// TIA Portal V17 export
// export: Created 2025-03-07T09:16:44.2659713Z, ExportSetting WithDefaults, DisplayName Totally Integrated Automation Portal, DisplayVersion V17 Update 8, DisplayName TIA Portal Openness, DisplayVersion V17 Update 8, DisplayName TIA Portal Version Control Interface, DisplayVersion V17, DisplayName SINAMICS Startdrive Advanced, DisplayVersion V17 SP2, DisplayName SINAMICS Startdrive G110M, G120, G120C, G120D, G120P, G115D, DisplayVersion V17 SP2, DisplayName SINAMICS Startdrive G130, G150, S120, S150, SINAMICS MV, S210, DisplayVersion V17 SP2, DisplayName STEP 7 Professional, DisplayVersion V17 Update 8, DisplayName SINUMERIK ONE STEP 7 Toolbox, DisplayVersion V17 Update 12, DisplayName SINUMERIK 840D sl STEP 7 Toolbox, DisplayVersion V17 Update 12, DisplayName STEP 7 Safety, DisplayVersion V17 Update 6, DisplayName WinCC Advanced, DisplayVersion V17 Update 8
FUNCTION "FC3001_JAW_CHUCK_CONTROL_U01_STA_1" : Void   // FC3001, LAD
{ S7_Optimized_Access := 'TRUE' }
VERSION : 0.1
// stored: AutoNumber false, IsIECCheckEnabled false, SetENOAutomatically false, UDAEnableTagReadback false
   VAR_TEMP
      TEMP_SENSOR_VALUE_1 : UInt;
      TEMP_SENSOR_VALUE : UInt;
   END_VAR
BEGIN

REGION Network 1: INPUTS
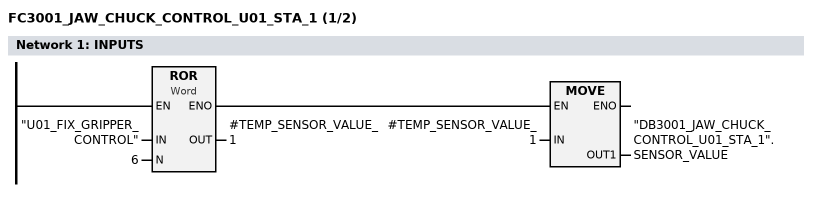
   #TEMP_SENSOR_VALUE_1 := ROR(IN := "U01_FIX_GRIPPER_CONTROL", N := 6);
   "DB3001_JAW_CHUCK_CONTROL_U01_STA_1".SENSOR_VALUE := #TEMP_SENSOR_VALUE_1;
END_REGION

REGION Network 2: UNIT 01 STATION 1 FIXTURE CLAMPED
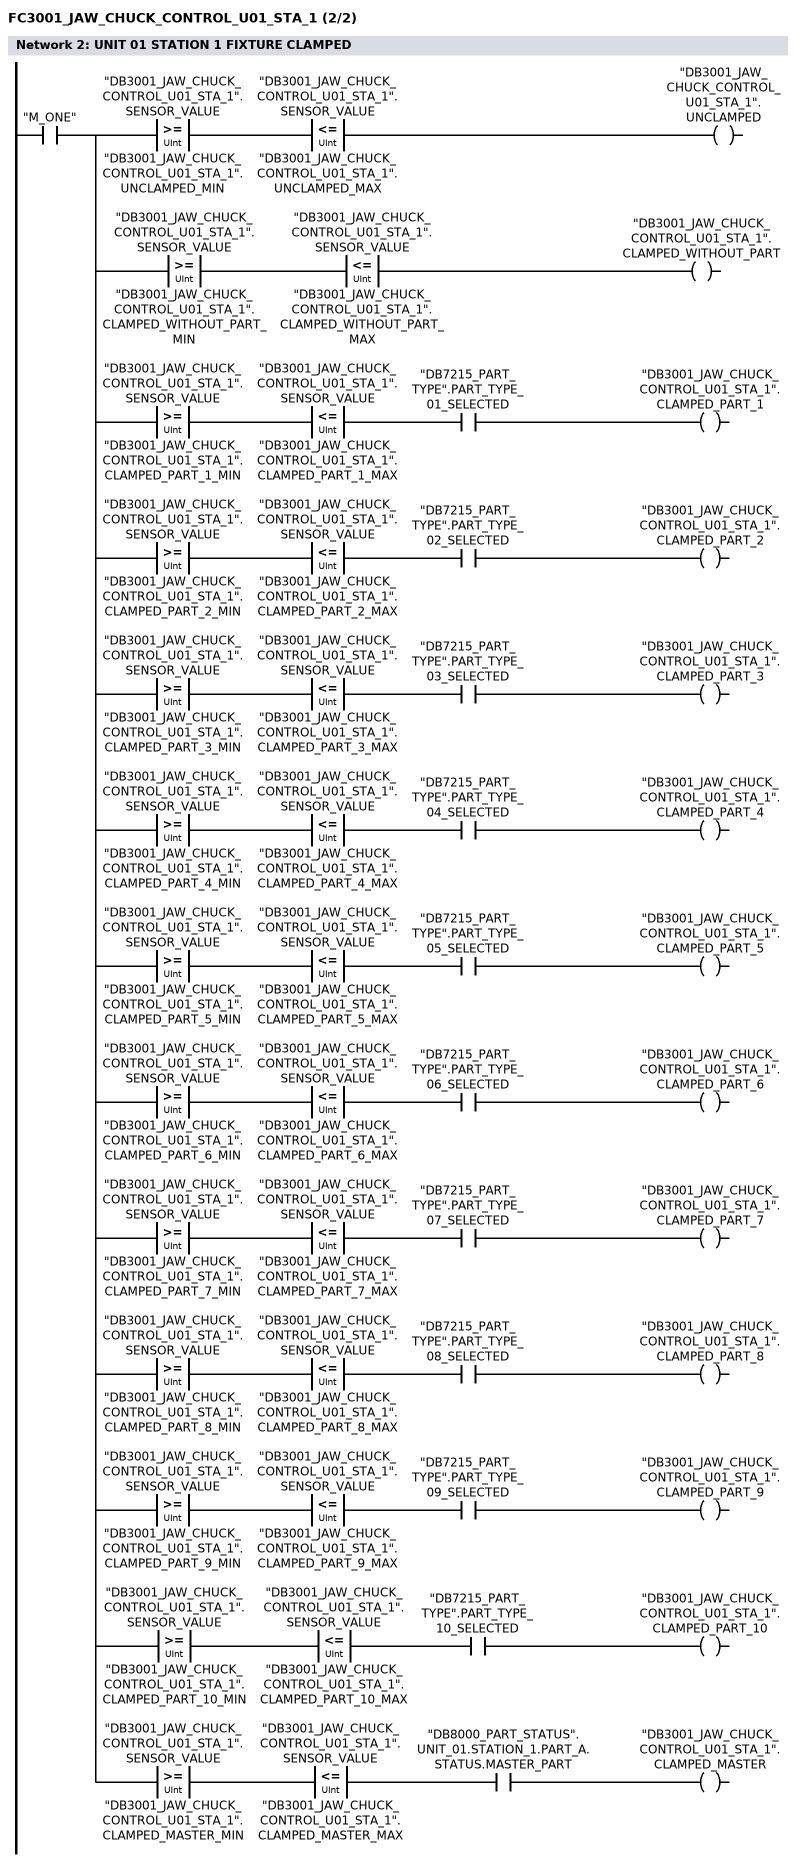
   RUNG wire#powerrail
      Contact( "M_ONE" )
      wire#w1
      { S7_Templates := "SrcType := UInt" } GE_Contact(in1 := "DB3001_JAW_CHUCK_CONTROL_U01_STA_1".SENSOR_VALUE, in2 := "DB3001_JAW_CHUCK_CONTROL_U01_STA_1".UNCLAMPED_MIN)
      { S7_Templates := "SrcType := UInt" } LE_Contact(in1 := "DB3001_JAW_CHUCK_CONTROL_U01_STA_1".SENSOR_VALUE, in2 := "DB3001_JAW_CHUCK_CONTROL_U01_STA_1".UNCLAMPED_MAX)
      Coil( "DB3001_JAW_CHUCK_CONTROL_U01_STA_1".UNCLAMPED )
   END_RUNG
   RUNG wire#w1
      { S7_Templates := "SrcType := UInt" } GE_Contact(in1 := "DB3001_JAW_CHUCK_CONTROL_U01_STA_1".SENSOR_VALUE, in2 := "DB3001_JAW_CHUCK_CONTROL_U01_STA_1".CLAMPED_WITHOUT_PART_MIN)
      { S7_Templates := "SrcType := UInt" } LE_Contact(in1 := "DB3001_JAW_CHUCK_CONTROL_U01_STA_1".SENSOR_VALUE, in2 := "DB3001_JAW_CHUCK_CONTROL_U01_STA_1".CLAMPED_WITHOUT_PART_MAX)
      Coil( "DB3001_JAW_CHUCK_CONTROL_U01_STA_1".CLAMPED_WITHOUT_PART )
   END_RUNG
   RUNG wire#w1
      { S7_Templates := "SrcType := UInt" } GE_Contact(in1 := "DB3001_JAW_CHUCK_CONTROL_U01_STA_1".SENSOR_VALUE, in2 := "DB3001_JAW_CHUCK_CONTROL_U01_STA_1".CLAMPED_PART_1_MIN)
      { S7_Templates := "SrcType := UInt" } LE_Contact(in1 := "DB3001_JAW_CHUCK_CONTROL_U01_STA_1".SENSOR_VALUE, in2 := "DB3001_JAW_CHUCK_CONTROL_U01_STA_1".CLAMPED_PART_1_MAX)
      Contact( "DB7215_PART_TYPE".PART_TYPE_01_SELECTED )
      Coil( "DB3001_JAW_CHUCK_CONTROL_U01_STA_1".CLAMPED_PART_1 )
   END_RUNG
   RUNG wire#w1
      { S7_Templates := "SrcType := UInt" } GE_Contact(in1 := "DB3001_JAW_CHUCK_CONTROL_U01_STA_1".SENSOR_VALUE, in2 := "DB3001_JAW_CHUCK_CONTROL_U01_STA_1".CLAMPED_PART_2_MIN)
      { S7_Templates := "SrcType := UInt" } LE_Contact(in1 := "DB3001_JAW_CHUCK_CONTROL_U01_STA_1".SENSOR_VALUE, in2 := "DB3001_JAW_CHUCK_CONTROL_U01_STA_1".CLAMPED_PART_2_MAX)
      Contact( "DB7215_PART_TYPE".PART_TYPE_02_SELECTED )
      Coil( "DB3001_JAW_CHUCK_CONTROL_U01_STA_1".CLAMPED_PART_2 )
   END_RUNG
   RUNG wire#w1
      { S7_Templates := "SrcType := UInt" } GE_Contact(in1 := "DB3001_JAW_CHUCK_CONTROL_U01_STA_1".SENSOR_VALUE, in2 := "DB3001_JAW_CHUCK_CONTROL_U01_STA_1".CLAMPED_PART_3_MIN)
      { S7_Templates := "SrcType := UInt" } LE_Contact(in1 := "DB3001_JAW_CHUCK_CONTROL_U01_STA_1".SENSOR_VALUE, in2 := "DB3001_JAW_CHUCK_CONTROL_U01_STA_1".CLAMPED_PART_3_MAX)
      Contact( "DB7215_PART_TYPE".PART_TYPE_03_SELECTED )
      Coil( "DB3001_JAW_CHUCK_CONTROL_U01_STA_1".CLAMPED_PART_3 )
   END_RUNG
   RUNG wire#w1
      { S7_Templates := "SrcType := UInt" } GE_Contact(in1 := "DB3001_JAW_CHUCK_CONTROL_U01_STA_1".SENSOR_VALUE, in2 := "DB3001_JAW_CHUCK_CONTROL_U01_STA_1".CLAMPED_PART_4_MIN)
      { S7_Templates := "SrcType := UInt" } LE_Contact(in1 := "DB3001_JAW_CHUCK_CONTROL_U01_STA_1".SENSOR_VALUE, in2 := "DB3001_JAW_CHUCK_CONTROL_U01_STA_1".CLAMPED_PART_4_MAX)
      Contact( "DB7215_PART_TYPE".PART_TYPE_04_SELECTED )
      Coil( "DB3001_JAW_CHUCK_CONTROL_U01_STA_1".CLAMPED_PART_4 )
   END_RUNG
   RUNG wire#w1
      { S7_Templates := "SrcType := UInt" } GE_Contact(in1 := "DB3001_JAW_CHUCK_CONTROL_U01_STA_1".SENSOR_VALUE, in2 := "DB3001_JAW_CHUCK_CONTROL_U01_STA_1".CLAMPED_PART_5_MIN)
      { S7_Templates := "SrcType := UInt" } LE_Contact(in1 := "DB3001_JAW_CHUCK_CONTROL_U01_STA_1".SENSOR_VALUE, in2 := "DB3001_JAW_CHUCK_CONTROL_U01_STA_1".CLAMPED_PART_5_MAX)
      Contact( "DB7215_PART_TYPE".PART_TYPE_05_SELECTED )
      Coil( "DB3001_JAW_CHUCK_CONTROL_U01_STA_1".CLAMPED_PART_5 )
   END_RUNG
   RUNG wire#w1
      { S7_Templates := "SrcType := UInt" } GE_Contact(in1 := "DB3001_JAW_CHUCK_CONTROL_U01_STA_1".SENSOR_VALUE, in2 := "DB3001_JAW_CHUCK_CONTROL_U01_STA_1".CLAMPED_PART_6_MIN)
      { S7_Templates := "SrcType := UInt" } LE_Contact(in1 := "DB3001_JAW_CHUCK_CONTROL_U01_STA_1".SENSOR_VALUE, in2 := "DB3001_JAW_CHUCK_CONTROL_U01_STA_1".CLAMPED_PART_6_MAX)
      Contact( "DB7215_PART_TYPE".PART_TYPE_06_SELECTED )
      Coil( "DB3001_JAW_CHUCK_CONTROL_U01_STA_1".CLAMPED_PART_6 )
   END_RUNG
   RUNG wire#w1
      { S7_Templates := "SrcType := UInt" } GE_Contact(in1 := "DB3001_JAW_CHUCK_CONTROL_U01_STA_1".SENSOR_VALUE, in2 := "DB3001_JAW_CHUCK_CONTROL_U01_STA_1".CLAMPED_PART_7_MIN)
      { S7_Templates := "SrcType := UInt" } LE_Contact(in1 := "DB3001_JAW_CHUCK_CONTROL_U01_STA_1".SENSOR_VALUE, in2 := "DB3001_JAW_CHUCK_CONTROL_U01_STA_1".CLAMPED_PART_7_MAX)
      Contact( "DB7215_PART_TYPE".PART_TYPE_07_SELECTED )
      Coil( "DB3001_JAW_CHUCK_CONTROL_U01_STA_1".CLAMPED_PART_7 )
   END_RUNG
   RUNG wire#w1
      { S7_Templates := "SrcType := UInt" } GE_Contact(in1 := "DB3001_JAW_CHUCK_CONTROL_U01_STA_1".SENSOR_VALUE, in2 := "DB3001_JAW_CHUCK_CONTROL_U01_STA_1".CLAMPED_PART_8_MIN)
      { S7_Templates := "SrcType := UInt" } LE_Contact(in1 := "DB3001_JAW_CHUCK_CONTROL_U01_STA_1".SENSOR_VALUE, in2 := "DB3001_JAW_CHUCK_CONTROL_U01_STA_1".CLAMPED_PART_8_MAX)
      Contact( "DB7215_PART_TYPE".PART_TYPE_08_SELECTED )
      Coil( "DB3001_JAW_CHUCK_CONTROL_U01_STA_1".CLAMPED_PART_8 )
   END_RUNG
   RUNG wire#w1
      { S7_Templates := "SrcType := UInt" } GE_Contact(in1 := "DB3001_JAW_CHUCK_CONTROL_U01_STA_1".SENSOR_VALUE, in2 := "DB3001_JAW_CHUCK_CONTROL_U01_STA_1".CLAMPED_PART_9_MIN)
      { S7_Templates := "SrcType := UInt" } LE_Contact(in1 := "DB3001_JAW_CHUCK_CONTROL_U01_STA_1".SENSOR_VALUE, in2 := "DB3001_JAW_CHUCK_CONTROL_U01_STA_1".CLAMPED_PART_9_MAX)
      Contact( "DB7215_PART_TYPE".PART_TYPE_09_SELECTED )
      Coil( "DB3001_JAW_CHUCK_CONTROL_U01_STA_1".CLAMPED_PART_9 )
   END_RUNG
   RUNG wire#w1
      { S7_Templates := "SrcType := UInt" } GE_Contact(in1 := "DB3001_JAW_CHUCK_CONTROL_U01_STA_1".SENSOR_VALUE, in2 := "DB3001_JAW_CHUCK_CONTROL_U01_STA_1".CLAMPED_PART_10_MIN)
      { S7_Templates := "SrcType := UInt" } LE_Contact(in1 := "DB3001_JAW_CHUCK_CONTROL_U01_STA_1".SENSOR_VALUE, in2 := "DB3001_JAW_CHUCK_CONTROL_U01_STA_1".CLAMPED_PART_10_MAX)
      Contact( "DB7215_PART_TYPE".PART_TYPE_10_SELECTED )
      Coil( "DB3001_JAW_CHUCK_CONTROL_U01_STA_1".CLAMPED_PART_10 )
   END_RUNG
   RUNG wire#w1
      { S7_Templates := "SrcType := UInt" } GE_Contact(in1 := "DB3001_JAW_CHUCK_CONTROL_U01_STA_1".SENSOR_VALUE, in2 := "DB3001_JAW_CHUCK_CONTROL_U01_STA_1".CLAMPED_MASTER_MIN)
      { S7_Templates := "SrcType := UInt" } LE_Contact(in1 := "DB3001_JAW_CHUCK_CONTROL_U01_STA_1".SENSOR_VALUE, in2 := "DB3001_JAW_CHUCK_CONTROL_U01_STA_1".CLAMPED_MASTER_MAX)
      Contact( "DB8000_PART_STATUS".UNIT_01.STATION_1.PART_A.STATUS.MASTER_PART )
      Coil( "DB3001_JAW_CHUCK_CONTROL_U01_STA_1".CLAMPED_MASTER )
   END_RUNG
   // the same network as SCL:
   "DB3001_JAW_CHUCK_CONTROL_U01_STA_1".UNCLAMPED := "M_ONE" AND ("DB3001_JAW_CHUCK_CONTROL_U01_STA_1".SENSOR_VALUE >= "DB3001_JAW_CHUCK_CONTROL_U01_STA_1".UNCLAMPED_MIN) AND ("DB3001_JAW_CHUCK_CONTROL_U01_STA_1".SENSOR_VALUE <= "DB3001_JAW_CHUCK_CONTROL_U01_STA_1".UNCLAMPED_MAX);
   "DB3001_JAW_CHUCK_CONTROL_U01_STA_1".CLAMPED_WITHOUT_PART := "M_ONE" AND ("DB3001_JAW_CHUCK_CONTROL_U01_STA_1".SENSOR_VALUE >= "DB3001_JAW_CHUCK_CONTROL_U01_STA_1".CLAMPED_WITHOUT_PART_MIN) AND ("DB3001_JAW_CHUCK_CONTROL_U01_STA_1".SENSOR_VALUE <= "DB3001_JAW_CHUCK_CONTROL_U01_STA_1".CLAMPED_WITHOUT_PART_MAX);
   "DB3001_JAW_CHUCK_CONTROL_U01_STA_1".CLAMPED_PART_1 := "M_ONE" AND ("DB3001_JAW_CHUCK_CONTROL_U01_STA_1".SENSOR_VALUE >= "DB3001_JAW_CHUCK_CONTROL_U01_STA_1".CLAMPED_PART_1_MIN) AND ("DB3001_JAW_CHUCK_CONTROL_U01_STA_1".SENSOR_VALUE <= "DB3001_JAW_CHUCK_CONTROL_U01_STA_1".CLAMPED_PART_1_MAX) AND "DB7215_PART_TYPE".PART_TYPE_01_SELECTED;
   "DB3001_JAW_CHUCK_CONTROL_U01_STA_1".CLAMPED_PART_2 := "M_ONE" AND ("DB3001_JAW_CHUCK_CONTROL_U01_STA_1".SENSOR_VALUE >= "DB3001_JAW_CHUCK_CONTROL_U01_STA_1".CLAMPED_PART_2_MIN) AND ("DB3001_JAW_CHUCK_CONTROL_U01_STA_1".SENSOR_VALUE <= "DB3001_JAW_CHUCK_CONTROL_U01_STA_1".CLAMPED_PART_2_MAX) AND "DB7215_PART_TYPE".PART_TYPE_02_SELECTED;
   "DB3001_JAW_CHUCK_CONTROL_U01_STA_1".CLAMPED_PART_3 := "M_ONE" AND ("DB3001_JAW_CHUCK_CONTROL_U01_STA_1".SENSOR_VALUE >= "DB3001_JAW_CHUCK_CONTROL_U01_STA_1".CLAMPED_PART_3_MIN) AND ("DB3001_JAW_CHUCK_CONTROL_U01_STA_1".SENSOR_VALUE <= "DB3001_JAW_CHUCK_CONTROL_U01_STA_1".CLAMPED_PART_3_MAX) AND "DB7215_PART_TYPE".PART_TYPE_03_SELECTED;
   "DB3001_JAW_CHUCK_CONTROL_U01_STA_1".CLAMPED_PART_4 := "M_ONE" AND ("DB3001_JAW_CHUCK_CONTROL_U01_STA_1".SENSOR_VALUE >= "DB3001_JAW_CHUCK_CONTROL_U01_STA_1".CLAMPED_PART_4_MIN) AND ("DB3001_JAW_CHUCK_CONTROL_U01_STA_1".SENSOR_VALUE <= "DB3001_JAW_CHUCK_CONTROL_U01_STA_1".CLAMPED_PART_4_MAX) AND "DB7215_PART_TYPE".PART_TYPE_04_SELECTED;
   "DB3001_JAW_CHUCK_CONTROL_U01_STA_1".CLAMPED_PART_5 := "M_ONE" AND ("DB3001_JAW_CHUCK_CONTROL_U01_STA_1".SENSOR_VALUE >= "DB3001_JAW_CHUCK_CONTROL_U01_STA_1".CLAMPED_PART_5_MIN) AND ("DB3001_JAW_CHUCK_CONTROL_U01_STA_1".SENSOR_VALUE <= "DB3001_JAW_CHUCK_CONTROL_U01_STA_1".CLAMPED_PART_5_MAX) AND "DB7215_PART_TYPE".PART_TYPE_05_SELECTED;
   "DB3001_JAW_CHUCK_CONTROL_U01_STA_1".CLAMPED_PART_6 := "M_ONE" AND ("DB3001_JAW_CHUCK_CONTROL_U01_STA_1".SENSOR_VALUE >= "DB3001_JAW_CHUCK_CONTROL_U01_STA_1".CLAMPED_PART_6_MIN) AND ("DB3001_JAW_CHUCK_CONTROL_U01_STA_1".SENSOR_VALUE <= "DB3001_JAW_CHUCK_CONTROL_U01_STA_1".CLAMPED_PART_6_MAX) AND "DB7215_PART_TYPE".PART_TYPE_06_SELECTED;
   "DB3001_JAW_CHUCK_CONTROL_U01_STA_1".CLAMPED_PART_7 := "M_ONE" AND ("DB3001_JAW_CHUCK_CONTROL_U01_STA_1".SENSOR_VALUE >= "DB3001_JAW_CHUCK_CONTROL_U01_STA_1".CLAMPED_PART_7_MIN) AND ("DB3001_JAW_CHUCK_CONTROL_U01_STA_1".SENSOR_VALUE <= "DB3001_JAW_CHUCK_CONTROL_U01_STA_1".CLAMPED_PART_7_MAX) AND "DB7215_PART_TYPE".PART_TYPE_07_SELECTED;
   "DB3001_JAW_CHUCK_CONTROL_U01_STA_1".CLAMPED_PART_8 := "M_ONE" AND ("DB3001_JAW_CHUCK_CONTROL_U01_STA_1".SENSOR_VALUE >= "DB3001_JAW_CHUCK_CONTROL_U01_STA_1".CLAMPED_PART_8_MIN) AND ("DB3001_JAW_CHUCK_CONTROL_U01_STA_1".SENSOR_VALUE <= "DB3001_JAW_CHUCK_CONTROL_U01_STA_1".CLAMPED_PART_8_MAX) AND "DB7215_PART_TYPE".PART_TYPE_08_SELECTED;
   "DB3001_JAW_CHUCK_CONTROL_U01_STA_1".CLAMPED_PART_9 := "M_ONE" AND ("DB3001_JAW_CHUCK_CONTROL_U01_STA_1".SENSOR_VALUE >= "DB3001_JAW_CHUCK_CONTROL_U01_STA_1".CLAMPED_PART_9_MIN) AND ("DB3001_JAW_CHUCK_CONTROL_U01_STA_1".SENSOR_VALUE <= "DB3001_JAW_CHUCK_CONTROL_U01_STA_1".CLAMPED_PART_9_MAX) AND "DB7215_PART_TYPE".PART_TYPE_09_SELECTED;
   "DB3001_JAW_CHUCK_CONTROL_U01_STA_1".CLAMPED_PART_10 := "M_ONE" AND ("DB3001_JAW_CHUCK_CONTROL_U01_STA_1".SENSOR_VALUE >= "DB3001_JAW_CHUCK_CONTROL_U01_STA_1".CLAMPED_PART_10_MIN) AND ("DB3001_JAW_CHUCK_CONTROL_U01_STA_1".SENSOR_VALUE <= "DB3001_JAW_CHUCK_CONTROL_U01_STA_1".CLAMPED_PART_10_MAX) AND "DB7215_PART_TYPE".PART_TYPE_10_SELECTED;
   "DB3001_JAW_CHUCK_CONTROL_U01_STA_1".CLAMPED_MASTER := "M_ONE" AND ("DB3001_JAW_CHUCK_CONTROL_U01_STA_1".SENSOR_VALUE >= "DB3001_JAW_CHUCK_CONTROL_U01_STA_1".CLAMPED_MASTER_MIN) AND ("DB3001_JAW_CHUCK_CONTROL_U01_STA_1".SENSOR_VALUE <= "DB3001_JAW_CHUCK_CONTROL_U01_STA_1".CLAMPED_MASTER_MAX) AND "DB8000_PART_STATUS".UNIT_01.STATION_1.PART_A.STATUS.MASTER_PART;
END_REGION
END_FUNCTION
